KUKA KRL data list: Psani.dat

&ACCESS RVO1
&REL 60
&PARAM EDITMASK = *
&PARAM TEMPLATE = C:\KRC\Roboter\Template\vorgabe
&PARAM DISKPATH = KRC:\R1\PPR\Psaci_Robot
DEFDAT  Psani
;FOLD EXTERNAL DECLARATIONS;%{PE}%MKUKATPBASIS,%CEXT,%VCOMMON,%P
;FOLD BASISTECH EXT;%{PE}%MKUKATPBASIS,%CEXT,%VEXT,%P
EXT  BAS (BAS_COMMAND  :IN,REAL  :IN )
DECL INT SUCCESS
;ENDFOLD (BASISTECH EXT)
;FOLD USER EXT;%{E}%MKUKATPUSER,%CEXT,%VEXT,%P
;Make your modifications here

;ENDFOLD (USER EXT)
;ENDFOLD (EXTERNAL DECLARATIONS)
DECL E6POS HomeBOD={X -11.6761513,Y -419.415039,Z 162.343185,A 91.4024582,B 28.6396141,C -179.395538,S 2,T 10,E1 0.0,E2 0.0,E3 0.0,E4 0.0,E5 0.0,E6 0.0}
DECL FRAME BOD={X 229.573853,Y -319.415039,Z 152.343185,A 91.4024582,B 28.6396141,C -179.395538}


ENDDAT
